FUNCTION_BLOCK MoveRelativeTask EXTENDS MotionTask
VAR
	_TargetDistance : LREAL;
	McMoveRelative	: ARRAY[0..1] OF MC_MoveRelative;
	Active			: UDINT;
    _McBufferMode	: MC_BufferMode;
	_MoveOptions	: ST_MoveOptions;
END_VAR

PROPERTY BufferMode : REFERENCE TO MC_BufferMode
GET
BufferMode REF= _McBufferMode;
END_GET
END_PROPERTY

{attribute 'monitoring' := 'call'}
PROPERTY Busy : BOOL
GET
Busy := McMoveRelative[Active].Busy;
END_GET
END_PROPERTY

METHOD CyclicLogic
VAR
    i : UDINT;
END_VAR
FOR i := 0 TO 1 DO
    McMoveRelative[i](Axis			:= _Axis.Axis,
                      Distance		:= _TargetDistance,
                      Velocity		:= _Axis.Velocity,
                      Acceleration := _Axis.Acceleration,
                      Deceleration := _Axis.Deceleration,
                      Jerk			:= _Axis.Jerk,
                      BufferMode	:= _McBufferMode,
                      Options		:= _MoveOptions);
    
    McMoveRelative[i].Execute := FALSE;
END_FOR
END_METHOD

{attribute 'monitoring' := 'call'}
PROPERTY Error : BOOL
GET
Error := McMoveRelative[Active].Error;
END_GET
END_PROPERTY

{attribute 'monitoring' := 'call'}
PROPERTY ErrorId : UDINT
GET
ErrorID := McMoveRelative[Active].ErrorID;
END_GET
END_PROPERTY

METHOD Execute : BOOL;
IF Active = 0 THEN
	Active := 1;
	McMoveRelative[Active](Axis			:= _Axis.Axis,
						   Execute		:= TRUE,
						   Distance		:= _TargetDistance,
						   Velocity		:= _Axis.Velocity,
						   Acceleration := _Axis.Acceleration,
						   Deceleration := _Axis.Deceleration,
						   Jerk			:= _Axis.Jerk,
						   BufferMode	:= _McBufferMode,
						   Options		:= _MoveOptions);
ELSE
	Active := 0;
	McMoveRelative[Active](Axis			:= _Axis.Axis,
						   Execute		:= TRUE,
						   Distance		:= _TargetDistance,
						   Velocity		:= _Axis.Velocity,
						   Acceleration := _Axis.Acceleration,
						   Deceleration := _Axis.Deceleration,
						   Jerk			:= _Axis.Jerk,
						   BufferMode	:= _McBufferMode,
						   Options		:= _MoveOptions);
END_IF

Execute := TRUE;
END_METHOD

PROPERTY MoveOptions : REFERENCE TO ST_MoveOptions
GET
MoveOptions REF= _MoveOptions;
END_GET
END_PROPERTY

{attribute 'monitoring' := 'call'}
PROPERTY TargetDistance : LREAL
SET
_TargetDistance := TargetDistance;
END_SET
END_PROPERTY

END_FUNCTION_BLOCK

(* stored: Version 1.1.0.1, ProductVersion 3.1.4026.18
   POU MoveRelativeTask: Id {3f565df6-70e4-4729-a1c3-76908c952c6a}, SpecialFunc None
   Property BufferMode: Id {fdf67959-47af-4d07-8e50-974781747229}
   Get Get: Id {9551f14c-5be9-4adf-b66a-fbafe73008ed}
   Property Busy: Id {346955dd-0ac4-4904-a668-cccb892d028f}
   Get Get: Id {76f96c15-1097-4fde-84db-0d65e7d0e9ed}
   Method CyclicLogic: Id {8a5fb35e-2a40-4f77-94a6-ccc71f19913b}
   Property Error: Id {10a364dc-ceca-48e6-ad8c-7020416da4d7}
   Get Get: Id {a5e83c72-636d-410f-8fc1-ba633837030d}
   Property ErrorId: Id {08704b46-ebd7-4455-8877-fe2723ecfdeb}
   Get Get: Id {26f7dd5e-4ad3-4b6c-88ac-a083091fe03b}
   Method Execute: Id {a63672ff-612b-4c36-9a37-963618bab1de}
   Property MoveOptions: Id {b2e19e7e-d653-4716-8dde-7931dc4b7083}
   Get Get: Id {6806118c-8733-4cd3-9c16-a47d7a9df5ab}
   Property TargetDistance: Id {0a515640-ffde-4942-a912-1fff5c7ef6dd}
   Set Set: Id {61eb5e6d-1c00-4f12-90b3-8f9a7fb160d7} *)
